ABB RobotStudio station: Project1.rsstnx

Station Project1 (saved by RobotStudio 26.3.11794.0)
Controller Controller36
  mechanical unit ROB_R: IRB14000_0.5_0.5_R, 6 joints, base frame (0, 0, 0) mm
  mechanical unit ROB_R_7: IRB14000_0.5_0.5_R, 1 joints, base frame (0, 0, 0) mm
  mechanical unit ROB_L: IRB14000_0.5_0.5_L, 6 joints, base frame (0, 0, 0) mm
  mechanical unit ROB_L_7: IRB14000_0.5_0.5_L, 1 joints, base frame (0, 0, 0) mm
Layout (positions relative to the parent item):
  - IRB14000_0.5_0.5 [mechanism, from %ABB.RobotStudio.Models.IRB14000%\IRB14000_0.5_0.5__02.rslib] at (0, 0, 0) mm
  - IRB14000_0.5_0.5_R [mechanism, from %ABB.RobotStudio.Models.IRB14000%\IRB14000_0.5_0.5__02.rslib] at (0, 0, 0) mm; joint values [1.2477, -2.4871, -1.2296, 0.872, -2.9466, 0.5122, 3.0778] (rad or m)
  - IRB14000_0.5_0.5_L [mechanism, from %ABB.RobotStudio.Models.IRB14000%\IRB14000_0.5_0.5__02.rslib] at (0, 0, 0) mm; joint values [-0.3837, -2.149, 1.1999, 0.4196, 0.4073, 0.6523, -1.2396] (rad or m)
  - Smart_Gripper_Servo_One_Vacuum_Fingers [mechanism, from %ABB.RobotStudio.Models.SmartGripper%\ABB_Smart_Gripper_Servo_One_Vacuum_Fingers.rslib] at (304.15, -157.57, 199.4) mm, rotated rx 178.73 ry -63.42 rz 15.81 deg; joint values [0] (rad or m)
  - Smart_Gripper_Servo_One_Vacuum_Camera_Fingers [mechanism, from %ABB.RobotStudio.Models.SmartGripper%\ABB_Smart_Gripper_Servo_One_Vacuum_Camera_Fingers.rslib] at (156.39, 439.53, 269.48) mm, rotated rx -179.34 ry -63.63 rz -15.45 deg; joint values [0] (rad or m)
  - SmartComponent_1 [smart component]
Attachment: Smart_Gripper_Servo_One_Vacuum_Fingers is attached to IRB14000_0.5_0.5_R / Link7
Attachment: Smart_Gripper_Servo_One_Vacuum_Camera_Fingers is attached to IRB14000_0.5_0.5_L / Link7
EventTableEntry 6498: ActivationMode=2, Cyclic=false, Group=, Trigger=do_openGrip 6499, Actions=[EventTableActionMechanicalPose 6500], Comment=
EventTableTriggerIO 6499: Operator=0, IOValue=[1], IRC5Controller=? -1, SignalSource=Controller36 3809
EventTableActionMechanicalPose 6500: VirtualSignal=, Mechanism=Smart_Gripper_Servo_One_Vacuum_Fingers 3786, ToPoseName=Position1, VirtualSignalValue=[1]
EventTableEntry 6501: ActivationMode=2, Cyclic=false, Group=, Trigger=do_openGrip 6502, Actions=[EventTableActionMechanicalPose 6503], Comment=
EventTableTriggerIO 6502: Operator=0, IOValue=[0], IRC5Controller=? -1, SignalSource=Controller36 3809
EventTableActionMechanicalPose 6503: VirtualSignal=, Mechanism=Smart_Gripper_Servo_One_Vacuum_Fingers 3786, ToPoseName=HomePosition, VirtualSignalValue=[1]
Station logic (signal -> signal, property => property):
  Controller36.do_openGrip -> Smart_Gripper_Servo_One_Vacuum_Camera_Fingers.Transform.X
Targets, tools, work objects and paths stored in the station, written as RAPID:
! task T_ROB_R
MODULE CalibData
  PERS tooldata Servo:=[TRUE,[[0,0,114.2],[1,0,0,0]],[0.226,[8.9,12.3,48.7],[1,0,0,0],0.00021,0.00024,0.00009]];
  PERS tooldata VaccumOne:=[TRUE,[[63.5,18.5,37.5],[0.707106781,0,0.707106781,0]],[0.226,[8.9,12.3,48.7],[1,0,0,0],0.00021,0.00024,0.00009]];
ENDMODULE

! task T_ROB_R
MODULE Module1
  CONST robtarget Home:=[[89.387946422,-156.622117956,147.913470217],[0.066010726,-0.842420918,-0.111214912,-0.523068661],[0,0,0,4],[-101.964427132,9E+09,9E+09,9E+09,9E+09,9E+09]];
ENDMODULE

! task T_ROB_L
MODULE CalibData
  PERS tooldata Servo:=[TRUE,[[0,0,114.2],[1,0,0,0]],[0.24,[8.2,12.5,48.1],[1,0,0,0],0.00022,0.00024,0.00009]];
  PERS tooldata VaccumOne:=[TRUE,[[63.5,18.5,37.5],[0.707106781,0,0.707106781,0]],[0.24,[8.2,12.5,48.1],[1,0,0,0],0.00022,0.00024,0.00009]];
  PERS tooldata Camera:=[TRUE,[[-7.3,28.3,35.1],[0.5,-0.5,0.5,0.5]],[0.24,[8.2,12.5,48.1],[1,0,0,0],0.00022,0.00024,0.00009]];
ENDMODULE

